Staubli VAL3: XHS3023L.pjx

--- XHS3023L.pjx ---
Parameters version=s7.7.2 stackSize=5000 millimeterUnit=true
Program file=loadNextOne.pgx
Program file=start.pgx
Program file=stop.pgx
Data file=XHS3023L.dtx
Library alias=prog path=.//XHS3023L1/XHS3023L1.pjx autoload=true password=
Library alias=prog_swap path=.//XHS3023L1/XHS3023L1.pjx autoload=true password=

--- XHS3023L.dtx ---
public frame fCadToReal = {fatherId=fUserFrame[0]}
public frame fUserFrame = {fatherId=world[0]}
public mdesc mNomSpeed = {blend=off}
public tool tTool = {x=968, y=-155, z=-238, rx=-90, rz=180, fatherId=flange[0], ioLink=valve1}

--- start.pgx ---
public program start()
begin

  prog:libLoad("Disk://XHS3023L/XHS3023L1")
  wait(taskStatus("loading")==-1)
  taskCreate "loading",10,loadNextOne("Disk://XHS3023L/XHS3023L2")
  call prog:start()

  prog:libLoad("Disk://XHS3023L/XHS3023L2")
  wait(taskStatus("loading")==-1)
  call prog:start()


end

--- loadNextOne.pgx ---
program loadNextOne(string x_sName (dimensions=1))
begin
  prog_swap:libLoad(x_sName)
end

--- stop.pgx ---
public program stop()
begin
  resetMotion()
end
